// TwinCAT 3 PLC project PcSpeaker_Player
// ProgramVersion: 3.1.4020.1
// libraries:
//   Tc2_Standard, * (Beckhoff Automation GmbH)
//   Tc2_System, * (Beckhoff Automation GmbH)
//   Tc3_Module, * (Beckhoff Automation GmbH)
//   Tc3_PcSpeaker, * (Nikolai Voronin)
// project tree:
//   GVLs/ Bach.TcGVL, Mario.TcGVL, StarWars.TcGVL
//   / PlcTask.TcTTO
//   POUs/ MAIN.TcPOU
// real-time tasks:
//   TASK PlcTask: cycle T#10ms, priority 20, ADS port 350

CONFIGURATION PcSpeaker_Player
    RESOURCE PLC ON TwinCAT3
        TASK PlcTask(INTERVAL := T#10ms, PRIORITY := 20);
        PROGRAM MAIN WITH PlcTask : MAIN;
    END_RESOURCE
END_CONFIGURATION

// ---- GVLs/Bach.TcGVL
{attribute 'qualified_only'}
VAR_GLOBAL CONSTANT
	BEEPS_MAX : UINT :=  1971;	
	Beeps : ARRAY[0..BEEPS_MAX] OF REAL := [98, 240, 0, 147, 240, 0, 247, 240, 0, 220, 240, 0, 247, 240, 0, 147, 240, 0, 247, 240, 0, 147, 240, 0, 98, 240, 0, 147, 240, 0, 247, 240, 0, 220, 240, 0, 247, 240, 0, 147, 240, 0, 247, 240, 0, 147, 240, 0, 98, 240, 0, 165, 240, 0, 262, 240, 0, 247, 240, 0, 262, 240, 0, 165, 240, 0, 262, 240, 0, 165, 240, 0, 98, 240, 0, 165, 240, 0, 262, 240, 0, 247, 240, 0, 262, 240, 0, 165, 240, 0, 262, 240, 0, 165, 240, 0, 98, 240, 0, 185, 240, 0, 262, 240, 0, 247, 240, 0, 262, 240, 0, 185, 240, 0, 262, 240, 0, 185, 240, 0, 98, 240, 0, 185, 240, 0, 262, 240, 0, 247, 240, 0, 262, 240, 0, 185, 240, 0, 262, 240, 0, 185, 240, 0, 98, 240, 0, 196, 240, 0, 247, 240, 0, 220, 240, 0, 247, 240, 0, 196, 240, 0, 247, 240, 0, 196, 240, 0, 98, 240, 0, 196, 240, 0, 247, 240, 0, 220, 240, 0, 247, 240, 0, 196, 240, 0, 247, 240, 0, 185, 240, 0, 98, 240, 0, 165, 240, 0, 247, 240, 0, 220, 240, 0, 247, 240, 0, 196, 240, 0, 185, 240, 0, 196, 240, 0, 165, 240, 0, 196, 240, 0, 185, 240, 0, 196, 240, 0, 123, 240, 0, 147, 240, 0, 139, 240, 0, 123, 240, 0, 139, 240, 0, 196, 240, 0, 220, 240, 0, 196, 240, 0, 220, 240, 0, 196, 240, 0, 220, 240, 0, 196, 240, 0, 139, 240, 0, 196, 240, 0, 220, 240, 0, 196, 240, 0, 220, 240, 0, 196, 240, 0, 220, 240, 0, 196, 240, 0, 185, 240, 0, 220, 240, 0, 294, 240, 0, 277, 240, 0, 294, 240, 0, 220, 240, 0, 196, 240, 0, 220, 240, 0, 185, 240, 0, 220, 240, 0, 196, 240, 0, 220, 240, 0, 147, 240, 0, 185, 240, 0, 165, 240, 0, 147, 240, 0, 82, 240, 0, 123, 240, 0, 196, 240, 0, 185, 240, 0, 196, 240, 0, 123, 240, 0, 196, 240, 0, 123, 240, 0, 82, 240, 0, 123, 240, 0, 196, 240, 0, 185, 240, 0, 196, 240, 0, 123, 240, 0, 196, 240, 0, 123, 240, 0, 82, 240, 0, 139, 240, 0, 147, 240, 0, 165, 240, 0, 147, 240, 0, 139, 240, 0, 123, 240, 0, 110, 240, 0, 196, 240, 0, 185, 240, 0, 165, 240, 0, 294, 240, 0, 277, 240, 0, 247, 240, 0, 220, 240, 0, 196, 240, 0, 185, 240, 0, 165, 240, 0, 147, 240, 0, 294, 240, 0, 220, 240, 0, 294, 240, 0, 185, 240, 0, 220, 240, 0, 147, 240, 0, 165, 240, 0, 185, 240, 0, 220, 240, 0, 196, 240, 0, 185, 240, 0, 165, 240, 0, 147, 240, 0, 208, 240, 0, 147, 240, 0, 175, 240, 0, 165, 240, 0, 175, 240, 0, 147, 240, 0, 208, 240, 0, 147, 240, 0, 247, 240, 0, 147, 240, 0, 175, 240, 0, 165, 240, 0, 175, 240, 0, 147, 240, 0, 208, 240, 0, 147, 240, 0, 131, 240, 0, 165, 240, 0, 220, 240, 0, 247, 240, 0, 262, 240, 0, 220, 240, 0, 165, 240, 0, 147, 240, 0, 131, 240, 0, 165, 240, 0, 220, 240, 0, 247, 240, 0, 262, 240, 0, 220, 240, 0, 185, 240, 0, 165, 240, 0, 156, 240, 0, 185, 240, 0, 156, 240, 0, 185, 240, 0, 220, 240, 0, 185, 240, 0, 220, 240, 0, 185, 240, 0, 156, 240, 0, 185, 240, 0, 156, 240, 0, 185, 240, 0, 220, 240, 0, 185, 240, 0, 220, 240, 0, 185, 240, 0, 196, 240, 0, 185, 240, 0, 165, 240, 0, 196, 240, 0, 185, 240, 0, 196, 240, 0, 220, 240, 0, 185, 240, 0, 196, 240, 0, 185, 240, 0, 165, 240, 0, 147, 240, 0, 131, 240, 0, 123, 240, 0, 110, 240, 0, 98, 240, 0, 92, 240, 0, 131, 240, 0, 147, 240, 0, 131, 240, 0, 147, 240, 0, 131, 240, 0, 147, 240, 0, 131, 240, 0, 92, 240, 0, 131, 240, 0, 147, 240, 0, 131, 240, 0, 147, 240, 0, 131, 240, 0, 147, 240, 0, 131, 240, 0, 98, 240, 0, 123, 240, 0, 175, 240, 0, 165, 240, 0, 175, 240, 0, 123, 240, 0, 175, 240, 0, 123, 240, 0, 98, 240, 0, 123, 240, 0, 175, 240, 0, 165, 240, 0, 175, 240, 0, 123, 240, 0, 175, 240, 0, 123, 240, 0, 98, 240, 0, 131, 240, 0, 165, 240, 0, 147, 240, 0, 165, 240, 0, 131, 240, 0, 165, 240, 0, 131, 240, 0, 98, 240, 0, 131, 240, 0, 165, 240, 0, 147, 240, 0, 165, 240, 0, 131, 240, 0, 165, 240, 0, 131, 240, 0, 98, 240, 0, 185, 240, 0, 262, 240, 0, 247, 240, 0, 262, 240, 0, 185, 240, 0, 262, 240, 0, 185, 240, 0, 98, 240, 0, 185, 240, 0, 262, 240, 0, 247, 240, 0, 262, 240, 0, 185, 240, 0, 262, 240, 0, 185, 240, 0, 98, 240, 0, 147, 240, 0, 247, 240, 0, 220, 240, 0, 247, 240, 0, 196, 240, 0, 185, 240, 0, 165, 240, 0, 147, 240, 0, 131, 240, 0, 123, 240, 0, 110, 240, 0, 98, 240, 0, 92, 240, 0, 82, 240, 0, 73, 240, 0, 69, 240, 0, 110, 240, 0, 165, 240, 0, 185, 240, 0, 196, 240, 0, 165, 240, 0, 185, 240, 0, 196, 240, 0, 69, 240, 0, 110, 240, 0, 165, 240, 0, 185, 240, 0, 196, 240, 0, 165, 240, 0, 185, 240, 0, 196, 240, 0, 65, 240, 0, 110, 240, 0, 147, 240, 0, 165, 240, 0, 185, 240, 0, 147, 240, 0, 165, 240, 0, 185, 240, 0, 65, 240, 0, 110, 240, 0, 147, 240, 0, 165, 240, 0, 185, 240, 0, 147, 240, 0, 165, 240, 0, 185, 240, 0, 65, 240, 0, 110, 240, 0, 147, 240, 0, 185, 240, 0, 220, 240, 0, 277, 240, 0, 294, 720, 0, 110, 240, 0, 123, 240, 0, 131, 240, 0, 147, 240, 0, 165, 240, 0, 185, 240, 0, 196, 240, 0, 220, 240, 0, 185, 240, 0, 147, 240, 0, 165, 240, 0, 185, 240, 0, 196, 240, 0, 220, 240, 0, 247, 240, 0, 262, 240, 0, 220, 240, 0, 185, 240, 0, 196, 240, 0, 220, 240, 0, 247, 240, 0, 262, 240, 0, 294, 240, 0, 311, 240, 0, 294, 240, 0, 277, 240, 0, 294, 240, 0, 294, 240, 0, 262, 240, 0, 247, 240, 0, 262, 240, 0, 262, 240, 0, 220, 240, 0, 185, 240, 0, 165, 240, 0, 147, 240, 0, 110, 240, 0, 123, 240, 0, 131, 240, 0, 73, 240, 0, 110, 240, 0, 147, 240, 0, 185, 240, 0, 220, 240, 0, 247, 240, 0, 262, 240, 0, 220, 240, 0, 247, 240, 0, 196, 240, 0, 147, 240, 0, 131, 240, 0, 123, 240, 0, 98, 240, 0, 110, 240, 0, 123, 240, 0, 73, 240, 0, 98, 240, 0, 123, 240, 0, 147, 240, 0, 196, 240, 0, 220, 240, 0, 247, 240, 0, 196, 240, 0, 277, 240, 0, 247, 240, 0, 220, 240, 0, 233, 240, 0, 233, 240, 0, 220, 240, 0, 208, 240, 0, 220, 240, 0, 220, 240, 0, 196, 240, 0, 185, 240, 0, 196, 240, 0, 196, 240, 0, 165, 240, 0, 139, 240, 0, 123, 240, 0, 110, 240, 0, 139, 240, 0, 165, 240, 0, 196, 240, 0, 220, 240, 0, 277, 240, 0, 294, 240, 0, 277, 240, 0, 294, 240, 0, 220, 240, 0, 185, 240, 0, 165, 240, 0, 185, 240, 0, 220, 240, 0, 147, 240, 0, 185, 240, 0, 110, 240, 0, 147, 240, 0, 139, 240, 0, 123, 240, 0, 110, 240, 0, 98, 240, 0, 92, 240, 0, 82, 240, 0, 73, 480, 0, 262, 240, 0, 247, 240, 0, 220, 240, 0, 196, 240, 0, 185, 240, 0, 165, 240, 0, 147, 240, 0, 262, 240, 0, 247, 240, 0, 220, 240, 0, 196, 240, 0, 185, 240, 0, 165, 240, 0, 147, 240, 0, 131, 240, 0, 247, 240, 0, 220, 240, 0, 196, 240, 0, 185, 240, 0, 165, 240, 0, 147, 240, 0, 131, 240, 0, 123, 240, 0, 220, 240, 0, 196, 240, 0, 185, 240, 0, 165, 240, 0, 147, 240, 0, 131, 240, 0, 123, 240, 0, 110, 240, 0, 196, 240, 0, 185, 240, 0, 165, 240, 0, 185, 240, 0, 147, 240, 0, 165, 240, 0, 185, 240, 0, 196, 240, 0, 165, 240, 0, 185, 240, 0, 147, 240, 0, 196, 240, 0, 165, 240, 0, 185, 240, 0, 147, 240, 0, 196, 240, 0, 165, 240, 0, 185, 240, 0, 147, 240, 0, 165, 240, 0, 185, 240, 0, 196, 240, 0, 220, 240, 0, 247, 240, 0, 147, 240, 0, 220, 240, 0, 247, 240, 0, 262, 240, 0, 147, 240, 0, 247, 240, 0, 262, 240, 0, 294, 240, 0, 247, 240, 0, 262, 240, 0, 247, 240, 0, 262, 240, 0, 220, 240, 0, 247, 240, 0, 220, 240, 0, 247, 240, 0, 196, 240, 0, 220, 240, 0, 196, 240, 0, 220, 240, 0, 185, 240, 0, 196, 240, 0, 185, 240, 0, 196, 240, 0, 165, 240, 0, 185, 240, 0, 147, 240, 0, 165, 240, 0, 175, 240, 0, 185, 240, 0, 196, 240, 0, 208, 240, 0, 220, 240, 0, 233, 240, 0, 247, 240, 0, 262, 240, 0, 277, 240, 0, 294, 240, 0, 311, 240, 0, 330, 240, 0, 349, 240, 0, 370, 240, 0, 392, 240, 0, 247, 240, 0, 147, 240, 0, 247, 240, 0, 392, 240, 0, 247, 240, 0, 392, 240, 0, 247, 240, 0, 392, 240, 0, 247, 240, 0, 147, 240, 0, 247, 240, 0, 392, 240, 0, 247, 240, 0, 392, 240, 0, 247, 240, 0, 392, 240, 0, 220, 240, 0, 147, 240, 0, 220, 240, 0, 392, 240, 0, 220, 240, 0, 392, 240, 0, 220, 240, 0, 392, 240, 0, 220, 240, 0, 147, 240, 0, 220, 240, 0, 392, 240, 0, 220, 240, 0, 392, 240, 0, 220, 240, 0, 370, 240, 0, 262, 240, 0, 147, 240, 0, 262, 240, 0, 370, 240, 0, 262, 240, 0, 370, 240, 0, 262, 240, 0, 370, 240, 0, 262, 240, 0, 147, 240, 0, 262, 240, 0, 370, 240, 0, 262, 240, 0, 370, 240, 0, 262, 240, 0, 392, 3840, 0, 220, 240, 0, 220, 240, 0, 220, 240, 0, 220, 240, 0, 220, 240, 0, 220, 240, 0, 220, 240, 0, 220, 240, 0, 220, 240, 0, 220, 240, 0, 220, 240, 0, 220, 240, 0, 220, 240, 0, 220, 240, 0, 220, 240, 0, 220, 240, 0, 220, 240, 0, 220, 240, 0, 220, 240, 0, 220, 240, 0, 220, 240, 0, 220, 240, 0, 220, 240, 0, 220, 240, 0, 220, 240, 0, 220, 240, 0, 220, 240, 0, 220, 240, 0, 220, 240, 0, 220, 240, 0, 220, 240, 0, 220, 240, 0, 220, 240, 0, 220, 240, 0, 220, 240, 0, 220, 240, 0, 220, 240, 0, 220, 240, 0, 220, 240, 0, 220, 240, 0, 220, 240, 0, 220, 240, 0, 220, 240, 0, 220, 240, 0, 220, 240, 0, 220, 240, 0, 220, 240, 0, 147, 240, 0, 147, 240, 0, 147, 240, 0, 147, 240, 0, 147, 240, 0, 147, 240, 0, 147, 240, 0, 147, 240, 0, 147, 240, 0, 147, 240, 0, 147, 240, 0, 147, 240, 0, 147, 240, 0, 147, 240, 0, 247, 3840, 0, 98, 3840, 0, 0, 0, 0];
END_VAR

// ---- GVLs/Mario.TcGVL
{attribute 'qualified_only'}
VAR_GLOBAL CONSTANT
(* Super Mario Brothers Overworld *)
	Beeps : ARRAY[0..3327] OF REAL := [146, 20, 0, 369, 20, 0, 659, 20, 47, 146, 20, 0, 369, 20, 0, 659, 20, 189, 146, 20, 0, 369, 20, 0, 659, 20, 190, 146, 20, 0, 369, 20, 0, 523, 20, 47, 146, 20, 0, 369, 20, 0, 659, 20, 190, 391, 20, 0, 493, 20, 0, 783, 20, 475, 195, 20, 0, 391, 20, 0, 195, 20, 0, 391, 20, 473, 195, 20, 0, 329, 20, 0, 523, 20, 332, 164, 20, 0, 261, 20, 0, 391, 20, 332, 130, 20, 0, 195, 20, 0, 329, 20, 332, 174, 20, 0, 261, 20, 0, 440, 20, 189, 195, 20, 0, 293, 20, 0, 493, 20, 189, 184, 20, 0, 277, 20, 0, 466, 20, 47, 174, 20, 0, 261, 20, 0, 440, 20, 190, 164, 20, 0, 261, 20, 0, 391, 20, 95, 261, 20, 0, 391, 20, 0, 659, 20, 95, 329, 20, 0, 493, 20, 0, 783, 20, 95, 349, 20, 0, 523, 20, 0, 880, 20, 190, 293, 20, 0, 440, 20, 0, 698, 20, 47, 329, 20, 0, 493, 20, 0, 783, 20, 189, 261, 20, 0, 440, 20, 0, 659, 20, 189, 220, 20, 0, 329, 20, 0, 523, 20, 47, 246, 20, 0, 349, 20, 0, 587, 20, 47, 195, 20, 0, 293, 20, 0, 493, 20, 332, 195, 20, 0, 329, 20, 0, 523, 20, 332, 164, 20, 0, 261, 20, 0, 391, 20, 332, 130, 20, 0, 195, 20, 0, 329, 20, 332, 174, 20, 0, 261, 20, 0, 440, 20, 189, 195, 20, 0, 293, 20, 0, 493, 20, 189, 184, 20, 0, 277, 20, 0, 466, 20, 47, 174, 20, 0, 261, 20, 0, 440, 20, 190, 164, 20, 0, 261, 20, 0, 391, 20, 95, 261, 20, 0, 391, 20, 0, 659, 20, 95, 329, 20, 0, 493, 20, 0, 783, 20, 95, 349, 20, 0, 523, 20, 0, 880, 20, 190, 293, 20, 0, 440, 20, 0, 698, 20, 47, 329, 20, 0, 493, 20, 0, 783, 20, 189, 261, 20, 0, 440, 20, 0, 659, 20, 189, 220, 20, 0, 329, 20, 0, 523, 20, 47, 246, 20, 0, 349, 20, 0, 587, 20, 47, 195, 20, 0, 293, 20, 0, 493, 20, 332, 130, 95, 190, 659, 20, 0, 783, 20, 0, 659, 20, 0, 783, 20, 47, 195, 20, 0, 622, 20, 0, 739, 20, 47, 587, 20, 0, 698, 20, 0, 587, 20, 0, 698, 20, 47, 493, 20, 0, 622, 20, 0, 493, 20, 0, 622, 20, 47, 261, 95, 47, 523, 20, 0, 659, 20, 0, 523, 20, 0, 659, 20, 47, 174, 95, 47, 329, 20, 0, 415, 20, 0, 329, 20, 0, 415, 20, 47, 349, 20, 0, 440, 20, 0, 349, 20, 0, 440, 20, 47, 261, 20, 0, 391, 20, 0, 523, 20, 47, 261, 95, 47, 261, 20, 0, 440, 20, 0, 261, 20, 0, 440, 20, 47, 174, 20, 0, 329, 20, 0, 523, 20, 47, 349, 20, 0, 587, 20, 0, 349, 20, 0, 587, 20, 47, 130, 95, 190, 659, 20, 0, 783, 20, 0, 659, 20, 0, 783, 20, 47, 164, 20, 0, 622, 20, 0, 739, 20, 47, 587, 20, 0, 698, 20, 0, 587, 20, 0, 698, 20, 47, 493, 20, 0, 622, 20, 0, 493, 20, 0, 622, 20, 47, 195, 95, 47, 261, 20, 0, 523, 20, 0, 659, 20, 189, 698, 20, 0, 783, 20, 0, 1046, 20, 189, 698, 20, 0, 783, 20, 0, 1046, 20, 47, 698, 20, 0, 783, 20, 0, 1046, 20, 190, 195, 95, 190, 130, 95, 190, 659, 20, 0, 783, 20, 0, 659, 20, 0, 783, 20, 47, 195, 20, 0, 622, 20, 0, 739, 20, 47, 587, 20, 0, 698, 20, 0, 587, 20, 0, 698, 20, 47, 493, 20, 0, 622, 20, 0, 493, 20, 0, 622, 20, 47, 261, 95, 47, 523, 20, 0, 659, 20, 0, 523, 20, 0, 659, 20, 47, 174, 95, 47, 329, 20, 0, 415, 20, 0, 329, 20, 0, 415, 20, 47, 349, 20, 0, 440, 20, 0, 349, 20, 0, 440, 20, 47, 261, 20, 0, 391, 20, 0, 523, 20, 47, 261, 95, 47, 261, 20, 0, 440, 20, 0, 261, 20, 0, 440, 20, 47, 174, 20, 0, 329, 20, 0, 523, 20, 47, 349, 20, 0, 587, 20, 0, 349, 20, 0, 587, 20, 47, 130, 95, 190, 207, 20, 0, 415, 20, 0, 622, 20, 332, 233, 20, 0, 349, 20, 0, 587, 20, 332, 261, 20, 0, 329, 20, 0, 523, 20, 332, 195, 94, 47, 195, 95, 190, 130, 95, 190, 130, 95, 190, 659, 20, 0, 783, 20, 0, 659, 20, 0, 783, 20, 47, 195, 20, 0, 622, 20, 0, 739, 20, 47, 587, 20, 0, 698, 20, 0, 587, 20, 0, 698, 20, 47, 493, 20, 0, 622, 20, 0, 493, 20, 0, 622, 20, 47, 261, 95, 47, 523, 20, 0, 659, 20, 0, 523, 20, 0, 659, 20, 47, 174, 95, 47, 329, 20, 0, 415, 20, 0, 329, 20, 0, 415, 20, 47, 349, 20, 0, 440, 20, 0, 349, 20, 0, 440, 20, 47, 261, 20, 0, 391, 20, 0, 523, 20, 47, 261, 95, 47, 261, 20, 0, 440, 20, 0, 261, 20, 0, 440, 20, 47, 174, 20, 0, 329, 20, 0, 523, 20, 47, 349, 20, 0, 587, 20, 0, 349, 20, 0, 587, 20, 47, 130, 95, 190, 659, 20, 0, 783, 20, 0, 659, 20, 0, 783, 20, 47, 164, 20, 0, 622, 20, 0, 739, 20, 47, 587, 20, 0, 698, 20, 0, 587, 20, 0, 698, 20, 47, 493, 20, 0, 622, 20, 0, 493, 20, 0, 622, 20, 47, 195, 95, 47, 261, 20, 0, 523, 20, 0, 659, 20, 189, 698, 20, 0, 783, 20, 0, 1046, 20, 189, 698, 20, 0, 783, 20, 0, 1046, 20, 47, 698, 20, 0, 783, 20, 0, 1046, 20, 190, 195, 95, 190, 130, 95, 190, 659, 20, 0, 783, 20, 0, 659, 20, 0, 783, 20, 47, 195, 20, 0, 622, 20, 0, 739, 20, 47, 587, 20, 0, 698, 20, 0, 587, 20, 0, 698, 20, 47, 493, 20, 0, 622, 20, 0, 493, 20, 0, 622, 20, 47, 261, 95, 47, 523, 20, 0, 659, 20, 0, 523, 20, 0, 659, 20, 47, 174, 95, 47, 329, 20, 0, 415, 20, 0, 329, 20, 0, 415, 20, 47, 349, 20, 0, 440, 20, 0, 349, 20, 0, 440, 20, 47, 261, 20, 0, 391, 20, 0, 523, 20, 47, 261, 95, 47, 261, 20, 0, 440, 20, 0, 261, 20, 0, 440, 20, 47, 174, 20, 0, 329, 20, 0, 523, 20, 47, 349, 20, 0, 587, 20, 0, 349, 20, 0, 587, 20, 47, 130, 95, 190, 207, 20, 0, 415, 20, 0, 622, 20, 332, 233, 20, 0, 349, 20, 0, 587, 20, 332, 261, 20, 0, 329, 20, 0, 523, 20, 332, 195, 94, 47, 195, 95, 190, 130, 95, 190, 103, 20, 0, 415, 20, 0, 523, 20, 47, 415, 20, 0, 523, 20, 0, 415, 20, 0, 523, 20, 189, 155, 20, 0, 415, 20, 0, 523, 20, 190, 415, 20, 0, 523, 20, 0, 415, 20, 0, 523, 20, 47, 207, 20, 0, 466, 20, 0, 587, 20, 190, 195, 20, 0, 391, 20, 0, 659, 20, 47, 329, 20, 0, 523, 20, 0, 329, 20, 0, 523, 20, 190, 130, 20, 0, 329, 20, 0, 440, 20, 47, 261, 20, 0, 391, 20, 0, 261, 20, 0, 391, 20, 189, 97, 95, 189, 103, 20, 0, 415, 20, 0, 523, 20, 47, 415, 20, 0, 523, 20, 0, 415, 20, 0, 523, 20, 189, 155, 20, 0, 415, 20, 0, 523, 20, 190, 415, 20, 0, 523, 20, 0, 415, 20, 0, 523, 20, 47, 207, 20, 0, 466, 20, 0, 587, 20, 47, 391, 20, 0, 659, 20, 0, 391, 20, 0, 659, 20, 47, 195, 95, 333, 130, 95, 332, 97, 95, 189, 103, 20, 0, 415, 20, 0, 523, 20, 47, 415, 20, 0, 523, 20, 0, 415, 20, 0, 523, 20, 189, 155, 20, 0, 415, 20, 0, 523, 20, 190, 415, 20, 0, 523, 20, 0, 415, 20, 0, 523, 20, 47, 207, 20, 0, 466, 20, 0, 587, 20, 190, 195, 20, 0, 391, 20, 0, 659, 20, 47, 329, 20, 0, 523, 20, 0, 329, 20, 0, 523, 20, 190, 130, 20, 0, 329, 20, 0, 440, 20, 47, 261, 20, 0, 391, 20, 0, 261, 20, 0, 391, 20, 189, 97, 95, 189, 146, 20, 0, 369, 20, 0, 659, 20, 47, 146, 20, 0, 369, 20, 0, 659, 20, 189, 146, 20, 0, 369, 20, 0, 659, 20, 190, 146, 20, 0, 369, 20, 0, 523, 20, 47, 146, 20, 0, 369, 20, 0, 659, 20, 190, 391, 20, 0, 493, 20, 0, 783, 20, 475, 195, 20, 0, 391, 20, 0, 195, 20, 0, 391, 20, 473, 195, 20, 0, 329, 20, 0, 523, 20, 332, 164, 20, 0, 261, 20, 0, 391, 20, 332, 130, 20, 0, 195, 20, 0, 329, 20, 332, 174, 20, 0, 261, 20, 0, 440, 20, 189, 195, 20, 0, 293, 20, 0, 493, 20, 189, 184, 20, 0, 277, 20, 0, 466, 20, 47, 174, 20, 0, 261, 20, 0, 440, 20, 190, 164, 20, 0, 261, 20, 0, 391, 20, 95, 261, 20, 0, 391, 20, 0, 659, 20, 95, 329, 20, 0, 493, 20, 0, 783, 20, 95, 349, 20, 0, 523, 20, 0, 880, 20, 190, 293, 20, 0, 440, 20, 0, 698, 20, 47, 329, 20, 0, 493, 20, 0, 783, 20, 189, 261, 20, 0, 440, 20, 0, 659, 20, 189, 220, 20, 0, 329, 20, 0, 523, 20, 47, 246, 20, 0, 349, 20, 0, 587, 20, 47, 195, 20, 0, 293, 20, 0, 493, 20, 332, 195, 20, 0, 329, 20, 0, 523, 20, 332, 164, 20, 0, 261, 20, 0, 391, 20, 332, 130, 20, 0, 195, 20, 0, 329, 20, 332, 174, 20, 0, 261, 20, 0, 440, 20, 189, 195, 20, 0, 293, 20, 0, 493, 20, 189, 184, 20, 0, 277, 20, 0, 466, 20, 47, 174, 20, 0, 261, 20, 0, 440, 20, 190, 164, 20, 0, 261, 20, 0, 391, 20, 95, 261, 20, 0, 391, 20, 0, 659, 20, 95, 329, 20, 0, 493, 20, 0, 783, 20, 95, 349, 20, 0, 523, 20, 0, 880, 20, 190, 293, 20, 0, 440, 20, 0, 698, 20, 47, 329, 20, 0, 493, 20, 0, 783, 20, 189, 261, 20, 0, 440, 20, 0, 659, 20, 189, 220, 20, 0, 329, 20, 0, 523, 20, 47, 246, 20, 0, 349, 20, 0, 587, 20, 47, 195, 20, 0, 293, 20, 0, 493, 20, 332, 130, 20, 0, 523, 20, 0, 659, 20, 47, 440, 20, 0, 523, 20, 0, 440, 20, 0, 523, 20, 190, 184, 20, 0, 329, 20, 0, 391, 20, 47, 195, 95, 190, 261, 20, 0, 329, 20, 0, 415, 20, 190, 174, 20, 0, 349, 20, 0, 440, 20, 47, 523, 20, 0, 698, 20, 0, 523, 20, 0, 698, 20, 47, 174, 95, 47, 523, 20, 0, 698, 20, 0, 523, 20, 0, 698, 20, 47, 261, 20, 0, 349, 20, 0, 440, 20, 47, 261, 94, 47, 174, 95, 190, 146, 20, 0, 391, 20, 0, 493, 20, 95, 698, 20, 0, 880, 20, 0, 698, 20, 0, 880, 20, 95, 698, 20, 0, 880, 20, 0, 174, 15, 0, 698, 15, 0, 880, 15, 0, 174, 47, 47, 195, 20, 0, 698, 20, 0, 880, 20, 95, 659, 20, 0, 783, 20, 0, 659, 20, 0, 783, 20, 0, 246, 95, 0, 587, 20, 0, 698, 20, 0, 587, 20, 0, 698, 20, 95, 195, 20, 0, 523, 20, 0, 659, 20, 47, 440, 20, 0, 523, 20, 0, 440, 20, 0, 523, 20, 47, 195, 95, 47, 349, 20, 0, 440, 20, 0, 349, 20, 0, 440, 20, 47, 261, 20, 0, 329, 20, 0, 391, 20, 47, 261, 94, 47, 195, 95, 190, 130, 20, 0, 523, 20, 0, 659, 20, 47, 440, 20, 0, 523, 20, 0, 440, 20, 0, 523, 20, 190, 184, 20, 0, 329, 20, 0, 391, 20, 47, 195, 95, 190, 261, 20, 0, 329, 20, 0, 415, 20, 190, 174, 20, 0, 349, 20, 0, 440, 20, 47, 523, 20, 0, 698, 20, 0, 523, 20, 0, 698, 20, 47, 174, 95, 47, 523, 20, 0, 698, 20, 0, 523, 20, 0, 698, 20, 47, 261, 20, 0, 349, 20, 0, 440, 20, 47, 261, 94, 47, 174, 95, 190, 195, 20, 0, 391, 20, 0, 493, 20, 47, 195, 20, 0, 587, 20, 0, 698, 20, 190, 195, 20, 0, 587, 20, 0, 698, 20, 47, 195, 20, 0, 587, 20, 0, 698, 20, 95, 220, 20, 0, 523, 20, 0, 659, 20, 95, 246, 20, 0, 493, 20, 0, 587, 20, 95, 261, 20, 0, 391, 20, 0, 523, 20, 47, 329, 95, 47, 195, 95, 47, 329, 95, 47, 130, 20, 0, 261, 20, 0, 130, 20, 0, 261, 20, 475, 130, 20, 0, 523, 20, 0, 659, 20, 47, 440, 20, 0, 523, 20, 0, 440, 20, 0, 523, 20, 190, 184, 20, 0, 329, 20, 0, 391, 20, 47, 195, 95, 190, 261, 20, 0, 329, 20, 0, 415, 20, 190, 174, 20, 0, 349, 20, 0, 440, 20, 47, 523, 20, 0, 698, 20, 0, 523, 20, 0, 698, 20, 47, 174, 95, 47, 523, 20, 0, 698, 20, 0, 523, 20, 0, 698, 20, 47, 261, 20, 0, 349, 20, 0, 440, 20, 47, 261, 94, 47, 174, 95, 190, 146, 20, 0, 391, 20, 0, 493, 20, 95, 698, 20, 0, 880, 20, 0, 698, 20, 0, 880, 20, 95, 698, 20, 0, 880, 20, 0, 174, 15, 0, 698, 15, 0, 880, 15, 0, 174, 47, 47, 195, 20, 0, 698, 20, 0, 880, 20, 95, 659, 20, 0, 783, 20, 0, 659, 20, 0, 783, 20, 0, 246, 95, 0, 587, 20, 0, 698, 20, 0, 587, 20, 0, 698, 20, 95, 195, 20, 0, 523, 20, 0, 659, 20, 47, 440, 20, 0, 523, 20, 0, 440, 20, 0, 523, 20, 47, 195, 95, 47, 349, 20, 0, 440, 20, 0, 349, 20, 0, 440, 20, 47, 261, 20, 0, 329, 20, 0, 391, 20, 47, 261, 94, 47, 195, 95, 190, 130, 20, 0, 523, 20, 0, 659, 20, 47, 440, 20, 0, 523, 20, 0, 440, 20, 0, 523, 20, 190, 184, 20, 0, 329, 20, 0, 391, 20, 47, 195, 95, 190, 261, 20, 0, 329, 20, 0, 415, 20, 190, 174, 20, 0, 349, 20, 0, 440, 20, 47, 523, 20, 0, 698, 20, 0, 523, 20, 0, 698, 20, 47, 174, 95, 47, 523, 20, 0, 698, 20, 0, 523, 20, 0, 698, 20, 47, 261, 20, 0, 349, 20, 0, 440, 20, 47, 261, 94, 47, 174, 95, 190, 195, 20, 0, 391, 20, 0, 493, 20, 47, 195, 20, 0, 587, 20, 0, 698, 20, 190, 195, 20, 0, 587, 20, 0, 698, 20, 47, 195, 20, 0, 587, 20, 0, 698, 20, 95, 220, 20, 0, 523, 20, 0, 659, 20, 95, 246, 20, 0, 493, 20, 0, 587, 20, 95, 261, 20, 0, 391, 20, 0, 523, 20, 47, 329, 95, 47, 195, 95, 47, 329, 95, 47, 130, 20, 0, 261, 20, 0, 130, 20, 0, 261, 20, 475, 103, 20, 0, 415, 20, 0, 523, 20, 47, 415, 20, 0, 523, 20, 0, 415, 20, 0, 523, 20, 189, 155, 20, 0, 415, 20, 0, 523, 20, 190, 415, 20, 0, 523, 20, 0, 415, 20, 0, 523, 20, 47, 207, 20, 0, 466, 20, 0, 587, 20, 190, 195, 20, 0, 391, 20, 0, 659, 20, 47, 329, 20, 0, 523, 20, 0, 329, 20, 0, 523, 20, 190, 130, 20, 0, 329, 20, 0, 440, 20, 47, 261, 20, 0, 391, 20, 0, 261, 20, 0, 391, 20, 189, 97, 95, 189, 103, 20, 0, 415, 20, 0, 523, 20, 47, 415, 20, 0, 523, 20, 0, 415, 20, 0, 523, 20, 189, 155, 20, 0, 415, 20, 0, 523, 20, 190, 415, 20, 0, 523, 20, 0, 415, 20, 0, 523, 20, 47, 207, 20, 0, 466, 20, 0, 587, 20, 47, 391, 20, 0, 659, 20, 0, 391, 20, 0, 659, 20, 47, 195, 95, 333, 130, 95, 332, 97, 95, 189, 103, 20, 0, 415, 20, 0, 523, 20, 47, 415, 20, 0, 523, 20, 0, 415, 20, 0, 523, 20, 189, 155, 20, 0, 415, 20, 0, 523, 20, 190, 415, 20, 0, 523, 20, 0, 415, 20, 0, 523, 20, 47, 207, 20, 0, 466, 20, 0, 587, 20, 190, 195, 20, 0, 391, 20, 0, 659, 20, 47, 329, 20, 0, 523, 20, 0, 329, 20, 0, 523, 20, 190, 130, 20, 0, 329, 20, 0, 440, 20, 47, 261, 20, 0, 391, 20, 0, 261, 20, 0, 391, 20, 189, 97, 95, 189, 146, 20, 0, 369, 20, 0, 659, 20, 47, 146, 20, 0, 369, 20, 0, 659, 20, 189, 146, 20, 0, 369, 20, 0, 659, 20, 190, 146, 20, 0, 369, 20, 0, 523, 20, 47, 146, 20, 0, 369, 20, 0, 659, 20, 190, 391, 20, 0, 493, 20, 0, 783, 20, 475, 195, 20, 0, 391, 20, 0, 195, 20, 0, 391, 20, 473, 130, 20, 0, 523, 20, 0, 659, 20, 47, 440, 20, 0, 523, 20, 0, 440, 20, 0, 523, 20, 190, 184, 20, 0, 329, 20, 0, 391, 20, 47, 195, 95, 190, 261, 20, 0, 329, 20, 0, 415, 20, 190, 174, 20, 0, 349, 20, 0, 440, 20, 47, 523, 20, 0, 698, 20, 0, 523, 20, 0, 698, 20, 47, 174, 95, 47, 523, 20, 0, 698, 20, 0, 523, 20, 0, 698, 20, 47, 261, 20, 0, 349, 20, 0, 440, 20, 47, 261, 94, 47, 174, 95, 190, 146, 20, 0, 391, 20, 0, 493, 20, 95, 698, 20, 0, 880, 20, 0, 698, 20, 0, 880, 20, 95, 698, 20, 0, 880, 20, 0, 174, 15, 0, 698, 15, 0, 880, 15, 0, 174, 47, 47, 195, 20, 0, 698, 20, 0, 880, 20, 95, 659, 20, 0, 783, 20, 0, 659, 20, 0, 783, 20, 0, 246, 95, 0, 587, 20, 0, 698, 20, 0, 587, 20, 0, 698, 20, 95, 195, 20, 0, 523, 20, 0, 659, 20, 47, 440, 20, 0, 523, 20, 0, 523, 20, 47, 195, 95, 47, 349, 20, 0, 440, 20, 0, 349, 20, 0, 440, 20, 47, 261, 20, 0, 329, 20, 0, 391, 20, 47, 261, 94, 47, 195, 95, 190, 130, 20, 0, 523, 20, 0, 659, 20, 47, 440, 20, 0, 523, 20, 0, 440, 20, 0, 523, 20, 190, 184, 20, 0, 329, 20, 0, 391, 20, 47, 195, 95, 190, 261, 20, 0, 329, 20, 0, 415, 20, 190, 174, 20, 0, 349, 20, 0, 440, 20, 47, 523, 20, 0, 698, 20, 0, 523, 20, 0, 698, 20, 47, 174, 95, 47, 523, 20, 0, 698, 20, 0, 523, 20, 0, 698, 20, 47, 261, 20, 0, 349, 20, 0, 440, 20, 47, 261, 94, 47, 174, 95, 190, 195, 20, 0, 391, 20, 0, 493, 20, 47, 195, 20, 0, 587, 20, 0, 698, 20, 190, 195, 20, 0, 587, 20, 0, 698, 20, 47, 195, 20, 0, 587, 20, 0, 698, 20, 95, 220, 20, 0, 523, 20, 0, 659, 20, 95, 246, 20, 0, 493, 20, 0, 587, 20, 95, 261, 20, 0, 391, 20, 0, 523, 20, 47, 329, 95, 47, 195, 95, 47, 329, 95, 47, 130, 20, 0, 261, 20, 0, 130, 20, 0, 261, 20, 0, 0, 0, 0];
END_VAR

// ---- GVLs/StarWars.TcGVL
{attribute 'qualified_only'}
VAR_GLOBAL CONSTANT
(* Star Wars Imperial March *) 
	Beeps : ARRAY[0..201] OF REAL := [392, 350, 100, 392, 350, 100, 392, 350, 100, 311, 250, 100, 466, 25, 100, 392, 350, 100, 311, 250, 100, 466, 25, 100, 392, 700, 100, 587, 350, 100, 587, 350, 100, 587, 350, 100, 622, 250, 100, 466, 25, 100, 369, 350, 100, 311, 250, 100, 466, 25, 100, 392, 700, 100, 784, 350, 100, 392, 250, 100, 392, 25, 100, 784, 350, 100, 739, 250, 100, 698, 25, 100, 659, 25, 100, 622, 25, 100, 659, 50, 400, 415, 25, 200, 554, 350, 100, 523, 250, 100, 493, 25, 100, 466, 25, 100, 440, 25, 100, 466, 50, 400, 311, 25, 200, 369, 350, 100, 311, 250, 100, 392, 25, 100, 466, 350, 100, 392, 250, 100, 466, 25, 100, 587, 700, 100, 784, 350, 100, 392, 250, 100, 392, 25, 100, 784, 350, 100, 739, 250, 100, 698, 25, 100, 659, 25, 100, 622, 25, 100, 659, 50, 400, 415, 25, 200, 554, 350, 100, 523, 250, 100, 493, 25, 100, 466, 25, 100, 440, 25, 100, 466, 50, 400, 311, 25, 200, 392, 350, 100, 311, 250, 100, 466, 25, 100, 392, 300, 150, 311, 250, 100, 466, 25, 100, 392, 700, 0, 0, 0, 0];
END_VAR

// ---- POUs/MAIN.TcPOU
PROGRAM MAIN
VAR
	START AT %I*	: BOOL;
	STOP AT %I*		: BOOL;

	Speaker	: FB_PcSpeaker;

	RTrig	: R_TRIG;
	state	: UINT;
	
	pNotes	: PVOID;
	F, L, D	: REAL;
	M		: REAL := 1; // duration multiplier
	szR		: UDINT := SIZEOF(REAL);
END_VAR

CASE state OF
0:
	RTrig(CLK := START);
	IF 	RTrig.Q THEN
		pNotes := ADR(StarWars.Beeps);	// <<<<<<<<<< Can change melody here
	
		START := FALSE;
		RTrig(CLK := FALSE);
		Speaker( Execute := FALSE );
		A_CopyNext();
		state := 100;
	END_IF

100: // Beep
	Speaker(
		Freq	:= REAL_TO_DWORD(F ),
		Length	:= REAL_TO_TIME( L * M ),
		Delay	:= REAL_TO_TIME( D ),
		Execute := TRUE );

	IF NOT Speaker.Busy THEN
		Speaker(Execute:= FALSE);
		A_CopyNext();
		IF (F = L) AND (L = D) AND (D = 0) THEN
			state := 0;
		END_IF
	END_IF

	RTrig(CLK := STOP);
	IF 	RTrig.Q THEN
		Speaker(Execute:= FALSE);
		Speaker.SwitchOff();
		STOP := FALSE;
		state := 0;
	END_IF
END_CASE

ACTION A_CopyNext:
MEMCPY(ADR(F), pNotes, szR);
pNotes := pNotes + szR;
MEMCPY(ADR(L), pNotes, szR);
pNotes := pNotes + szR;
MEMCPY(ADR(D), pNotes, szR);
pNotes := pNotes + szR;
END_ACTION

END_PROGRAM
